FUNCTION_BLOCK FB_FT_DERIV (* calculates the derivate over the signal in with Faktor K *)
  (* Standard: OSCAT; Classification: Control *)
  (* Version 0.0, 2011-07-04, 4DIAC-IDE, 4DIAC-Consortium *)
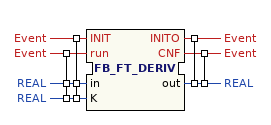
  EVENT_INPUT
    INIT WITH in, K; (* Initialization Request *)
    run WITH in, K; (* Normal Execution Request *)
  END_EVENT
  EVENT_OUTPUT
    INITO WITH out; (* Initialization Confirm *)
    CNF WITH out; (* Execution Confirmation *)
  END_EVENT
  VAR_INPUT
    in : REAL; (* Input signal *)
    K : REAL := 1.0; (* Factor *)
  END_VAR
  VAR_OUTPUT
    out : REAL; (* Result of the derivate *)
  END_VAR
  VAR
    old : REAL;
    tx : DWORD;
    last : DWORD;
    tc : REAL;
  END_VAR
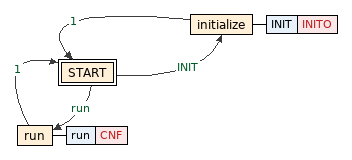
  EC_STATES
    START; (* Initial State *)
    initialize : INIT -> INITO; (* Initialization *)
    run : run -> CNF; (* Normal execution *)
  END_STATES
  EC_TRANSITIONS
    START TO initialize := INIT;
    initialize TO START := 1;
    START TO run := run;
    run TO START := 1;
  END_TRANSITIONS
  ALGORITHM INIT IN AnyText: (* Initialization algorithm *)
old() = in();
  END_ALGORITHM
  ALGORITHM run IN AnyText: (* Normally executed algorithm *)
tx() = T_PLC_US();
tc() = DWORD_TO_REAL(tx() - last());
last() = tx();

if(tc() > 0.0){
	out() = (in() - old()) / tc() * 1000000.0 * K();
	old() = in();
}else{
	out() = 0.0;
}
  END_ALGORITHM
END_FUNCTION_BLOCK
